Fanuc TP program (LS listing): _ati_lock.ls

/PROG  _ATI_LOCK	  Macro
/ATTR
OWNER		= MNEDITOR;
COMMENT		= "";
PROG_SIZE	= 203;
CREATE		= DATE 21-08-19  TIME 21:16:00;
MODIFIED	= DATE 21-08-19  TIME 21:16:00;
FILE_NAME	= ;
VERSION		= 0;
LINE_COUNT	= 3;
MEMORY_SIZE	= 563;
PROTECT		= READ_WRITE;
TCD:  STACK_SIZE	= 0,
      TASK_PRIORITY	= 50,
      TIME_SLICE	= 0,
      BUSY_LAMP_OFF	= 0,
      ABORT_REQUEST	= 0,
      PAUSE_REQUEST	= 0;
DEFAULT_GROUP	= *,*,*,*,*;
CONTROL_CODE	= 00000000 00000000;
/APPL
/APPL

AUTO_SINGULARITY_HEADER;
  ENABLE_SINGULARITY_AVOIDANCE   : TRUE;
/MN
   1:  DO[2:UNLOCK_TOOL]=OFF ;
   2:  DO[1:LOCK_TOOL]=ON ;
   3:  WAIT    .50(sec) ;
/POS
/END
